ABB RAPID module: Module1.mod

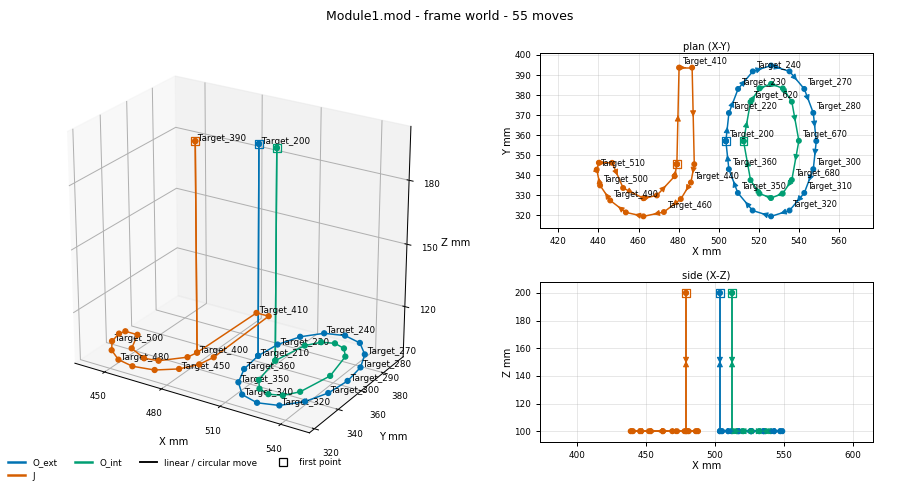
[picture p0: tool path of Module1.mod in frame world, 55 of 60 moves have a stored position in this frame; points joined in program order, loops and branches not executed]
MODULE Module1
    CONST robtarget Target_200:=[[-746.362477268,402.442634407,126.110538385],[0.382682909,0.923878273,-0.001525788,0.000632003],[0,0,0,0],[9E+09,9E+09,9E+09,9E+09,9E+09,9E+09]];
    CONST robtarget Target_210:=[[-746.362477268,331.731956437,55.399860119],[0.382682909,0.923878273,-0.001525788,0.000632003],[0,0,0,0],[9E+09,9E+09,9E+09,9E+09,9E+09,9E+09]];
    CONST robtarget Target_220:=[[-744.835979572,341.650188095,45.481628503],[0.38268291,0.923878273,-0.001525788,0.000632002],[0,0,0,0],[9E+09,9E+09,9E+09,9E+09,9E+09,9E+09]];
    CONST robtarget Target_230:=[[-740.256486485,350.142801239,36.989015393],[0.38268291,0.923878273,-0.001525788,0.000632002],[0,0,0,0],[9E+09,9E+09,9E+09,9E+09,9E+09,9E+09]];
    CONST robtarget Target_240:=[[-732.912016438,356.344241773,30.787574886],[0.38268291,0.923878273,-0.001525788,0.000632003],[0,0,0,0],[9E+09,9E+09,9E+09,9E+09,9E+09,9E+09]];
    CONST robtarget Target_250:=[[-723.781832107,358.411388617,28.72042805],[0.38268291,0.923878273,-0.001525788,0.000632002],[0,0,0,0],[9E+09,9E+09,9E+09,9E+09,9E+09,9E+09]];
    CONST robtarget Target_260:=[[-714.565242245,356.344241773,30.787574886],[0.38268291,0.923878273,-0.001525788,0.000632002],[0,0,0,0],[9E+09,9E+09,9E+09,9E+09,9E+09,9E+09]];
    CONST robtarget Target_270:=[[-707.191970356,350.142801239,36.989015393],[0.38268291,0.923878273,-0.001525788,0.000632002],[0,0,0,0],[9E+09,9E+09,9E+09,9E+09,9E+09,9E+09]];
    CONST robtarget Target_280:=[[-702.698882798,341.690920052,45.440896545],[0.38268291,0.923878273,-0.001525788,0.000632002],[0,0,0,0],[9E+09,9E+09,9E+09,9E+09,9E+09,9E+09]];
    CONST robtarget Target_290:=[[-701.201186945,331.731956437,55.399860119],[0.382682909,0.923878273,-0.001525788,0.000632003],[0,0,0,0],[9E+09,9E+09,9E+09,9E+09,9E+09,9E+09]];
    CONST robtarget Target_300:=[[-702.698882798,321.7933588,65.338457713],[0.38268291,0.923878273,-0.001525788,0.000632002],[0,0,0,0],[9E+09,9E+09,9E+09,9E+09,9E+09,9E+09]];
    CONST robtarget Target_310:=[[-707.191970356,313.40257555,73.729240928],[0.38268291,0.923878273,-0.001525788,0.000632002],[0,0,0,0],[9E+09,9E+09,9E+09,9E+09,9E+09,9E+09]];
    CONST robtarget Target_320:=[[-714.565242245,307.201135016,79.930681436],[0.38268291,0.923878273,-0.001525788,0.000632003],[0,0,0,0],[9E+09,9E+09,9E+09,9E+09,9E+09,9E+09]];
    CONST robtarget Target_330:=[[-723.781832107,305.133988171,81.997828272],[0.38268291,0.923878273,-0.001525788,0.000632002],[0,0,0,0],[9E+09,9E+09,9E+09,9E+09,9E+09,9E+09]];
    CONST robtarget Target_340:=[[-732.998421968,307.201135016,79.930681436],[0.38268291,0.923878273,-0.001525788,0.000632002],[0,0,0,0],[9E+09,9E+09,9E+09,9E+09,9E+09,9E+09]];
    CONST robtarget Target_350:=[[-740.371693858,313.40257555,73.729240928],[0.38268291,0.923878273,-0.001525788,0.000632002],[0,0,0,0],[9E+09,9E+09,9E+09,9E+09,9E+09,9E+09]];
    CONST robtarget Target_360:=[[-744.864781415,321.7933588,65.338457713],[0.38268291,0.923878273,-0.001525788,0.000632002],[0,0,0,0],[9E+09,9E+09,9E+09,9E+09,9E+09,9E+09]];
    CONST robtarget Target_370:=[[-746.362477268,331.731956437,55.399860119],[0.382682909,0.923878273,-0.001525788,0.000632003],[0,0,0,0],[9E+09,9E+09,9E+09,9E+09,9E+09,9E+09]];
    CONST robtarget Target_380:=[[-746.362477268,402.442634407,126.110538385],[0.382682909,0.923878273,-0.001525788,0.000632003],[0,0,0,0],[9E+09,9E+09,9E+09,9E+09,9E+09,9E+09]];
    CONST robtarget Target_390:=[[-770.844044088,394.255510945,134.297661814],[0.382682909,0.923878273,-0.001525788,0.000632002],[0,0,0,0],[9E+09,9E+09,9E+09,9E+09,9E+09,9E+09]];
    CONST robtarget Target_400:=[[-770.844044088,323.544832974,63.586983547],[0.382682909,0.923878273,-0.001525788,0.000632002],[0,0,0,0],[9E+09,9E+09,9E+09,9E+09,9E+09,9E+09]];
    CONST robtarget Target_410:=[[-769.749574042,357.668030393,29.463786272],[0.38268291,0.923878273,-0.001525788,0.000632002],[0,0,0,0],[9E+09,9E+09,9E+09,9E+09,9E+09,9E+09]];
    CONST robtarget Target_420:=[[-763.225956531,357.668030393,29.463786272],[0.382682909,0.923878273,-0.001525788,0.000632002],[0,0,0,0],[9E+09,9E+09,9E+09,9E+09,9E+09,9E+09]];
    CONST robtarget Target_430:=[[-762.145887406,323.544832974,63.586983547],[0.382682909,0.923878273,-0.001525788,0.000632002],[0,0,0,0],[9E+09,9E+09,9E+09,9E+09,9E+09,9E+09]];
    CONST robtarget Target_440:=[[-763.83079524,317.088817705,70.042998788],[0.382682909,0.923878273,-0.001525788,0.000632002],[0,0,0,0],[9E+09,9E+09,9E+09,9E+09,9E+09,9E+09]];
    CONST robtarget Target_450:=[[-768.885518743,311.243781801,75.888034669],[0.382682909,0.923878273,-0.001525788,0.000632002],[0,0,0,0],[9E+09,9E+09,9E+09,9E+09,9E+09,9E+09]];
    CONST robtarget Target_460:=[[-777.324458835,306.661436579,80.470379871],[0.382682909,0.923878273,-0.001525788,0.000632002],[0,0,0,0],[9E+09,9E+09,9E+09,9E+09,9E+09,9E+09]];
    CONST robtarget Target_470:=[[-787.549113213,305.133988171,81.997828272],[0.38268291,0.923878273,-0.001525788,0.000632002],[0,0,0,0],[9E+09,9E+09,9E+09,9E+09,9E+09,9E+09]];
    CONST robtarget Target_480:=[[-796.333675425,306.539240706,80.592575743],[0.38268291,0.923878273,-0.001525788,0.000632002],[0,0,0,0],[9E+09,9E+09,9E+09,9E+09,9E+09,9E+09]];
    CONST robtarget Target_490:=[[-804.138974964,310.75499831,76.376818157],[0.38268291,0.923878273,-0.001525788,0.000632002],[0,0,0,0],[9E+09,9E+09,9E+09,9E+09,9E+09,9E+09]];
    CONST robtarget Target_500:=[[-809.193698466,316.060335778,71.071480711],[0.382682909,0.923878273,-0.001525788,0.000632002],[0,0,0,0],[9E+09,9E+09,9E+09,9E+09,9E+09,9E+09]];
    CONST robtarget Target_510:=[[-810.8786063,321.63043097,65.501385543],[0.382682909,0.923878273,-0.001525788,0.000632002],[0,0,0,0],[9E+09,9E+09,9E+09,9E+09,9E+09,9E+09]];
    CONST robtarget Target_520:=[[-809.812938097,324.074348422,63.057468102],[0.38268291,0.923878273,-0.001525788,0.000632002],[0,0,0,0],[9E+09,9E+09,9E+09,9E+09,9E+09,9E+09]];
    CONST robtarget Target_530:=[[-803.202915056,324.043799454,63.08801707],[0.382682909,0.923878273,-0.001525788,0.000632002],[0,0,0,0],[9E+09,9E+09,9E+09,9E+09,9E+09,9E+09]];
    CONST robtarget Target_540:=[[-797.687362061,315.154049723,71.977766762],[0.38268291,0.923878273,-0.001525788,0.000632002],[0,0,0,0],[9E+09,9E+09,9E+09,9E+09,9E+09,9E+09]];
    CONST robtarget Target_550:=[[-787.549113213,311.528905504,75.602910967],[0.38268291,0.923878273,-0.001525788,0.000632002],[0,0,0,0],[9E+09,9E+09,9E+09,9E+09,9E+09,9E+09]];
    CONST robtarget Target_560:=[[-780.83828372,312.516655474,74.615161002],[0.38268291,0.923878273,-0.001525788,0.000632003],[0,0,0,0],[9E+09,9E+09,9E+09,9E+09,9E+09,9E+09]];
    CONST robtarget Target_570:=[[-771.967315978,319.308709391,67.823107112],[0.38268291,0.923878273,-0.001525788,0.000632002],[0,0,0,0],[9E+09,9E+09,9E+09,9E+09,9E+09,9E+09]];
    CONST robtarget Target_580:=[[-770.844044088,323.544832974,63.586983547],[0.382682909,0.923878273,-0.001525788,0.000632002],[0,0,0,0],[9E+09,9E+09,9E+09,9E+09,9E+09,9E+09]];
    CONST robtarget Target_590:=[[-770.844044088,394.255510945,134.297661814],[0.382682909,0.923878273,-0.001525788,0.000632002],[0,0,0,0],[9E+09,9E+09,9E+09,9E+09,9E+09,9E+09]];
    CONST robtarget Target_600:=[[-737.549113213,402.442634407,126.110538385],[0.382682909,0.923878273,-0.001525788,0.000632002],[0,0,0,0],[9E+09,9E+09,9E+09,9E+09,9E+09,9E+09]];
    CONST robtarget Target_610:=[[-737.549113213,331.731956437,55.399860119],[0.382682909,0.923878273,-0.001525788,0.000632002],[0,0,0,0],[9E+09,9E+09,9E+09,9E+09,9E+09,9E+09]];
    CONST robtarget Target_620:=[[-734.035288328,345.540090038,41.591726575],[0.38268291,0.923878273,-0.001525788,0.000632003],[0,0,0,0],[9E+09,9E+09,9E+09,9E+09,9E+09,9E+09]];
    CONST robtarget Target_630:=[[-729.571002614,350.336278037,36.795538596],[0.38268291,0.923878273,-0.001525788,0.000632002],[0,0,0,0],[9E+09,9E+09,9E+09,9E+09,9E+09,9E+09]];
    CONST robtarget Target_640:=[[-723.781832107,351.935007371,35.19680927],[0.38268291,0.923878273,-0.001525788,0.000632002],[0,0,0,0],[9E+09,9E+09,9E+09,9E+09,9E+09,9E+09]];
    CONST robtarget Target_650:=[[-717.90625607,350.356644016,36.775172617],[0.382682909,0.923878273,-0.001525788,0.000632002],[0,0,0,0],[9E+09,9E+09,9E+09,9E+09,9E+09,9E+09]];
    CONST robtarget Target_660:=[[-713.413168512,345.621553953,41.51026266],[0.38268291,0.923878273,-0.001525788,0.000632002],[0,0,0,0],[9E+09,9E+09,9E+09,9E+09,9E+09,9E+09]];
    CONST robtarget Target_670:=[[-709.899343627,331.813420352,55.318396204],[0.382682909,0.923878273,-0.001525788,0.000632002],[0,0,0,0],[9E+09,9E+09,9E+09,9E+09,9E+09,9E+09]];
    CONST robtarget Target_680:=[[-713.413168512,318.00528675,69.126529747],[0.38268291,0.923878273,-0.001525788,0.000632003],[0,0,0,0],[9E+09,9E+09,9E+09,9E+09,9E+09,9E+09]];
    CONST robtarget Target_690:=[[-717.963859756,313.209098751,73.922717726],[0.382682909,0.923878273,-0.001525788,0.000632002],[0,0,0,0],[9E+09,9E+09,9E+09,9E+09,9E+09,9E+09]];
    CONST robtarget Target_700:=[[-723.781832107,311.610369419,75.521447053],[0.38268291,0.923878273,-0.001525788,0.000632002],[0,0,0,0],[9E+09,9E+09,9E+09,9E+09,9E+09,9E+09]];
    CONST robtarget Target_710:=[[-729.571002614,313.188732772,73.943083705],[0.382682909,0.923878273,-0.001525788,0.000632002],[0,0,0,0],[9E+09,9E+09,9E+09,9E+09,9E+09,9E+09]];
    CONST robtarget Target_720:=[[-734.035288328,317.923822835,69.207993662],[0.38268291,0.923878273,-0.001525788,0.000632002],[0,0,0,0],[9E+09,9E+09,9E+09,9E+09,9E+09,9E+09]];
    CONST robtarget Target_730:=[[-737.549113213,331.731956437,55.399860119],[0.382682909,0.923878273,-0.001525788,0.000632002],[0,0,0,0],[9E+09,9E+09,9E+09,9E+09,9E+09,9E+09]];
    CONST robtarget Target_740:=[[-737.549113213,402.442634407,126.110538385],[0.382682909,0.923878273,-0.001525788,0.000632002],[0,0,0,0],[9E+09,9E+09,9E+09,9E+09,9E+09,9E+09]];
    CONST jointtarget home:=[[0,0,0,0,30.000000835,0],[9E+09,9E+09,9E+09,9E+09,9E+09,9E+09]];
    CONST jointtarget GoHome:=[[0,0,0,0,30,0],[9E+09,9E+09,9E+09,9E+09,9E+09,9E+09]];
    CONST jointtarget Homeoficial:=[[0,0,0,0,0,0],[9E+09,9E+09,9E+09,9E+09,9E+09,9E+09]];
    CONST jointtarget Mantenimiento:=[[-90,0,0,0,-30,0],[9E+09,9E+09,9E+09,9E+09,9E+09,9E+09]];
    CONST jointtarget JointTarget_2:=[[20.782622689,27.408337335,0,0,30,0],[9E+09,9E+09,9E+09,9E+09,9E+09,9E+09]];
!***********************************************************
    !
    ! Módulo:  Module1
    !
    ! Descripción:
    !   <Introduzca la descripción aquí>
    !
    ! Autor: Juan Andres
    !
    ! Versión: 1.0
    !
    !***********************************************************


    !***********************************************************
    !
    ! Procedimiento Main
    !
    !   Este es el punto de entrada de su programa
    !
    !***********************************************************
    PROC main()
       GoHome1 ;
       WaitDI Entrada1,1;
       SetDO Salida1,1;
       acercamiento ;
        J;
        O_ext;
        O_int;
        GoHome1;
        WaitDI Entrada2,1;
        SetDO Salida1,0;
        Out;
    ENDPROC

    PROC O_ext()
        SingArea \Wrist;
        ConfL \Off;
        MoveL Target_200,v50,z40,marcador_0\WObj:=Tablero;
        MoveL Target_210,v50,z5,marcador_0\WObj:=Tablero;
        MoveL Target_220,v50,z5,marcador_0\WObj:=Tablero;
        MoveL Target_230,v50,z5,marcador_0\WObj:=Tablero;
        MoveL Target_240,v50,z1,marcador_0\WObj:=Tablero;
        MoveL Target_250,v50,z1,marcador_0\WObj:=Tablero;
        MoveL Target_260,v50,z1,marcador_0\WObj:=Tablero;
        MoveL Target_270,v50,z5,marcador_0\WObj:=Tablero;
        MoveL Target_280,v50,z5,marcador_0\WObj:=Tablero;
        MoveL Target_290,v50,z5,marcador_0\WObj:=Tablero;
        MoveL Target_300,v50,z5,marcador_0\WObj:=Tablero;
        MoveL Target_310,v50,z5,marcador_0\WObj:=Tablero;
        MoveL Target_320,v50,z1,marcador_0\WObj:=Tablero;
        MoveL Target_330,v50,z1,marcador_0\WObj:=Tablero;
        MoveL Target_340,v50,z1,marcador_0\WObj:=Tablero;
        MoveL Target_350,v50,z5,marcador_0\WObj:=Tablero;
        MoveL Target_360,v50,z5,marcador_0\WObj:=Tablero;
        MoveL Target_370,v50,z5,marcador_0\WObj:=Tablero;
        MoveL Target_380,v50,z40,marcador_0\WObj:=Tablero;
    ENDPROC
    PROC J()
        SingArea \Wrist;
        ConfL \Off;
        MoveL Target_390,v50,z40,marcador_0\WObj:=Tablero;
        MoveL Target_400,v50,z20,marcador_0\WObj:=Tablero;
        MoveL Target_410,v50,z1,marcador_0\WObj:=Tablero;
        MoveL Target_420,v50,z1,marcador_0\WObj:=Tablero;
        MoveL Target_430,v50,z1,marcador_0\WObj:=Tablero;
        MoveL Target_440,v50,z1,marcador_0\WObj:=Tablero;
        MoveL Target_450,v50,z1,marcador_0\WObj:=Tablero;
        MoveL Target_460,v50,z5,marcador_0\WObj:=Tablero;
        MoveL Target_470,v50,z1,marcador_0\WObj:=Tablero;
        MoveL Target_480,v50,z1,marcador_0\WObj:=Tablero;
        MoveL Target_490,v50,z1,marcador_0\WObj:=Tablero;
        MoveL Target_500,v50,z1,marcador_0\WObj:=Tablero;
        MoveL Target_510,v50,z1,marcador_0\WObj:=Tablero;
        MoveL Target_520,v50,z1,marcador_0\WObj:=Tablero;
        MoveL Target_530,v50,z1,marcador_0\WObj:=Tablero;
        MoveL Target_540,v50,z5,marcador_0\WObj:=Tablero;
        MoveL Target_550,v50,z1,marcador_0\WObj:=Tablero;
        MoveL Target_560,v50,z1,marcador_0\WObj:=Tablero;
        MoveL Target_570,v50,z1,marcador_0\WObj:=Tablero;
        MoveL Target_580,v50,z1,marcador_0\WObj:=Tablero;
        MoveL Target_590,v50,z50,marcador_0\WObj:=Tablero;
    ENDPROC

    PROC GoHome1()
        MoveAbsJ GoHome,v1000,z100,marcador_0\WObj:=Tablero;
    ENDPROC


    PROC Out()

        MoveAbsJ home,v1000,z100,marcador_0\WObj:=Tablero;
        MoveAbsJ Mantenimiento,v1000,z100,marcador_0\WObj:=Tablero;
    ENDPROC
    PROC O_int()
        SingArea \Wrist;
        ConfL \Off;
        MoveL Target_600,v50,z40,marcador_0\WObj:=Tablero;
        MoveL Target_610,v50,z5,marcador_0\WObj:=Tablero;
        MoveL Target_620,v50,z1,marcador_0\WObj:=Tablero;
        MoveL Target_630,v50,z1,marcador_0\WObj:=Tablero;
        MoveL Target_640,v50,z1,marcador_0\WObj:=Tablero;
        MoveL Target_650,v50,z1,marcador_0\WObj:=Tablero;
        MoveL Target_660,v50,z1,marcador_0\WObj:=Tablero;
        MoveL Target_670,v50,z5,marcador_0\WObj:=Tablero;
        MoveL Target_680,v50,z1,marcador_0\WObj:=Tablero;
        MoveL Target_690,v50,z1,marcador_0\WObj:=Tablero;
        MoveL Target_700,v50,z1,marcador_0\WObj:=Tablero;
        MoveL Target_710,v50,z1,marcador_0\WObj:=Tablero;
        MoveL Target_720,v50,z1,marcador_0\WObj:=Tablero;
        MoveL Target_730,v50,z5,marcador_0\WObj:=Tablero;
        MoveL Target_740,v50,z40,marcador_0\WObj:=Tablero;
    ENDPROC
    PROC Home_30()
        MoveAbsJ home,v1000,z100,marcador_0\WObj:=Tablero;
    ENDPROC
    PROC acercamiento()
        MoveAbsJ JointTarget_2,v1000,z100,marcador_0\WObj:=Tablero;
    ENDPROC
ENDMODULE
